Fanuc KAREL source: kt00474.KL

PROGRAM KT00474
%STACKSIZE=65535
%PRIORITY=65535
%NOLOCKGROUP
VAR
P1 : POSITION
P2 : POSITION
OUT : POSITION
BEGIN
-- UNRESOLVED_PC line 8 opcodes [49 49 60 4A] marker_code=0
END KT00474
